INTERFACE I_MessageData

PROPERTY DirRoot : POINTER to string(255)
SET
END_SET
END_PROPERTY

PROPERTY ErrorIndex : reference to uint
SET
END_SET
END_PROPERTY

PROPERTY FileRoot : pointer to string(255)
SET
END_SET
END_PROPERTY

PROPERTY LocalTime : pointer to DT
SET
END_SET
END_PROPERTY

PROPERTY MessageIndex : reference to uint
SET
END_SET
END_PROPERTY

PROPERTY MsgList : pointer to ARRAY[1..GVL_MSG_XTS.MAX_MESSAGE] OF st_message
SET
END_SET
END_PROPERTY

END_INTERFACE

(* stored: Version 1.1.0.1
   Itf I_MessageData: Id {08f9e9aa-de9f-40c5-8536-4fe3cbec264d}
   Property DirRoot: Id {5e2f1e50-98ed-4923-bb25-ee09dd96e31c}
   Set Set: Id {2fd45f5f-e100-4257-9df7-e38cd3090ac1}
   Property ErrorIndex: Id {bd9261a0-3775-4ef6-b603-bd46850487ad}
   Set Set: Id {7728f7fd-a457-41bd-8691-8fa49d6c774b}
   Property FileRoot: Id {9bfe3fd9-ae24-4a39-9f95-e876e6ba1453}
   Set Set: Id {c57f2e86-0c42-451b-8870-2fcd11efea08}
   Property LocalTime: Id {1ccbaeb0-2164-4faa-a1c4-a1bee5cdb38d}
   Set Set: Id {50f784b5-a546-4507-bf23-174c15b93b13}
   Property MessageIndex: Id {f57ae467-6c6c-4170-9afb-17a73d17c3fe}
   Set Set: Id {29a2f697-ce50-4f05-b0c8-84d535a9efb7}
   Property MsgList: Id {c74b315f-0644-43bc-930b-3abff830c3ea}
   Set Set: Id {439a424c-273d-4a82-ae52-ac51e02a5999} *)
